(*
SPDX-FileCopyrightText: © 2026 Oleksandr Tiutyk <trofimich@gmail.com>
SPDX-License-Identifier: MIT
License: https://opensource.org/license/mit
*)

INTERFACE IGenericValueValidator EXTENDS IObject

METHOD Validate
VAR_INPUT
	validatedObjectName : WSTRING;
END_VAR
VAR_IN_OUT CONSTANT
	valueToValidate : GENERIC_VALUE;
END_VAR
END_METHOD

END_INTERFACE

(* stored: Version 1.1.0.1
   Itf IGenericValueValidator: Id {7dad695e-3ff1-4d4a-a4f7-428b8a6f5965}
   Method Validate: Id {e910886f-ea56-48f1-bf3c-15978736c0be} *)
